{attribute 'reflection'}
FUNCTION_BLOCK ABSTRACT FB_OrphanObject IMPLEMENTS I_Object
VAR
    _nIdentity:         ULINT;
    _ipSelf:            I_Object;

    {attribute 'instance-path'}
    {attribute 'noinit'}
    _sPath:             STRING(MAX_STRING_LENGTH);
END_VAR

PROPERTY bOrphan : BOOL
GET
bOrphan := TRUE;
END_GET
END_PROPERTY

METHOD Equals : BOOL
VAR_INPUT
    ipObject:       I_Object;
END_VAR
Equals := ipObject = THIS^._ipSelf;
END_METHOD

METHOD FB_init : BOOL
VAR_INPUT
    bInitRetains:           BOOL; // if TRUE, the retain variables are initialized (warm start / cold start)
    bInCopyCode:            BOOL;  // if TRUE, the instance afterwards gets moved into the copy code (online change)
END_VAR
_nIdentity := ADR(THIS^);
END_METHOD

PROPERTY ipContext : I_Context
GET
END_GET
END_PROPERTY

PROPERTY nIdentity : ULINT
GET
THIS^._nIdentity := ADR(THIS^);
nIdentity := THIS^._nIdentity;
END_GET
END_PROPERTY

PROPERTY sPath : STRING(MAX_STRING_LENGTH)
GET
sPath := THIS^._sPath;
END_GET
END_PROPERTY

END_FUNCTION_BLOCK

(* stored: Version 1.1.0.1, ProductVersion 3.1.4024.12
   POU FB_OrphanObject: Id {9656be67-d383-42c6-84f7-0402b86c0719}, SpecialFunc None
   Property bOrphan: Id {95212aa0-ae69-49d2-b8c4-dd0b74f3dd44}
   Get Get: Id {a7509e69-c338-4a17-826e-50c2b4a521f1}
   Method Equals: Id {271de0b5-8583-0d64-0611-ec8b4394066f}
   Method FB_init: Id {23c93e36-e082-4b93-a8b6-b4afc1cc1bc0}
   Property ipContext: Id {dffb61fc-8261-476e-8380-13ae59770e1d}
   Get Get: Id {bdcc517e-eead-457c-9ed9-d53ccb44e672}
   Property nIdentity: Id {6142e4e4-ee68-4eb6-a1fe-e30ec06c3e81}
   Get Get: Id {a5be8550-84e9-4c42-839d-1a284c4431b1}
   Property sPath: Id {1bc2a9e9-9f83-4b1a-92be-77e550760d9f}
   Get Get: Id {a1cd70cc-57fe-4a45-8b1f-64130ce7b943} *)
